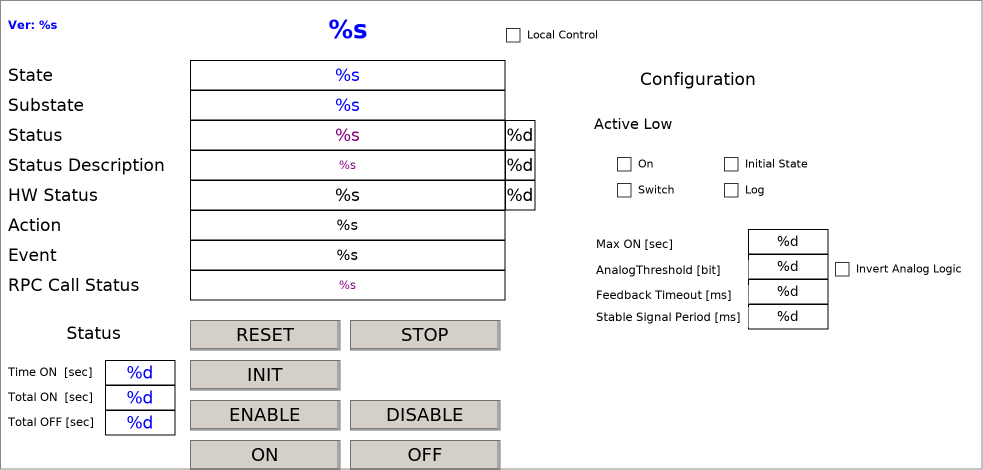
VISUALIZATION GUI_TEMPLATE_ACTUATOR  // 983x470
VAR_IN_OUT
	m_Instance:	FB_ACTUATOR;
END_VAR
    Rectangle (190,60 315x30), "%s", text variable: m_Instance.stat.sState
    Rectangle (190,90 315x30), "%s", text variable: m_Instance.stat.sSubstate
    Button (190,320 150x30), "RESET", input disabled if: (m_Instance.stat.bLocal = FALSE) <> 0
        OnMouseDown: execute { m_Instance.ctrl.nCommand := E_ACTUATOR_COMMAND.RESET; m_Instance.ctrl.bExecute := TRUE; }
    Button (190,360 150x30), "INIT", input disabled if: (m_Instance.stat.bLocal = FALSE) <> 0
        OnMouseDown: execute { m_Instance.ctrl.nCommand := E_ACTUATOR_COMMAND.INIT; m_Instance.ctrl.bExecute := TRUE; }
    Button (350,320 150x30), "STOP", input disabled if: (m_Instance.stat.bLocal = FALSE) <> 0
        OnMouseDown: execute { m_Instance.ctrl.nCommand := E_ACTUATOR_COMMAND.STOP; m_Instance.ctrl.bExecute := TRUE; }
    Button (190,400 150x30), "ENABLE", input disabled if: (m_Instance.stat.bLocal = FALSE) <> 0
        OnMouseDown: execute { m_Instance.ctrl.nCommand := E_ACTUATOR_COMMAND.ENABLE; m_Instance.ctrl.bExecute := TRUE; }
    Button (350,400 150x30), "DISABLE", input disabled if: (m_Instance.stat.bLocal = FALSE) <> 0
        OnMouseDown: execute { m_Instance.ctrl.nCommand := E_ACTUATOR_COMMAND.DISABLE; m_Instance.ctrl.bExecute := TRUE; }
    Button (190,440 150x30), "ON", input disabled if: (m_Instance.stat.bLocal = FALSE) <> 0
        OnMouseDown: execute { m_Instance.ctrl.nCommand := E_ACTUATOR_COMMAND.ON; m_Instance.ctrl.bExecute := TRUE; }
    Button (350,440 150x30), "OFF", input disabled if: (m_Instance.stat.bLocal = FALSE) <> 0
        OnMouseDown: execute { m_Instance.ctrl.nCommand := E_ACTUATOR_COMMAND.OFF; m_Instance.ctrl.bExecute := TRUE; }
    Rectangle (5,60 180x30), "State"
    Rectangle (5,90 180x30), "Substate"
    Rectangle (190,120 315x30), "%s", text variable: m_Instance.stat.sStatus
    Rectangle (190,150 315x30), "%s", text variable: m_Instance.stat.sErrorText
    Rectangle (5,120 180x30), "Status"
    Rectangle (5,150 180x30), "Status Description"
    Rectangle (190,210 315x30), "%s", text variable: m_Instance.stat.sActionDesc
    Rectangle (190,240 315x30), "%s", text variable: m_Instance.stat.sEventDesc
    Rectangle (190,180 315x30), "%s", text variable: m_Instance.stat.sHwStatus
    Rectangle (5,180 180x30), "HW Status"
    Rectangle (505,180 30x30), "%d", text variable: m_Instance.stat.nHwStatus
    Rectangle (5,210 180x30), "Action"
    Rectangle (5,240 180x30), "Event"
    Rectangle (232,12 232x35), "%s", text variable: m_Instance.cfg.sName
    Rectangle (637,64 180x30), "Configuration"
    Rectangle (591,109 126x30), "Active Low"
    Checkbox (615,149 72x30), "On", variable: m_Instance.cfg.bActiveLowOn, input disabled if: (m_Instance.stat.bLocal = FALSE) <> 0
    Checkbox (615,175 72x30), "Switch", variable: m_Instance.cfg.bActiveLowSwitch, input disabled if: (m_Instance.stat.bLocal = FALSE) <> 0
    Checkbox (833,254 150x30), "Invert Analog Logic", tooltip "If the logic is inverted, the actuator is considered to be ON, if the reading is below the threshold.", variable: m_Instance.cfg.bInvertAnalog, input disabled if: (m_Instance.stat.bLocal = FALSE) <> 0
    Rectangle (593,234 155x20), "Max ON [sec]"
    Rectangle (748,229 80x25), "%d", tooltip "Maximum allowed time for actuator to be ON [sec] (>=0). Zero means no limit.", text variable: m_Instance.cfg.nMaxOn, input disabled if: (m_Instance.stat.bLocal = FALSE) <> 0
        OnMouseDown: write the text variable via Default, min 0
    Rectangle (748,254 80x25), "%d", tooltip "Analog feedback signal threshold [bit]. If used, the threshold should be > 0.", text variable: m_Instance.cfg.nAnalogThreshold, input disabled if: (m_Instance.stat.bLocal = FALSE) <> 0
        OnMouseDown: write the text variable via Default, min 0
    Rectangle (593,260 155x20), "AnalogThreshold [bit]"
    Rectangle (748,279 80x25), "%d", tooltip "When switching actuator ON, feedback signal should become active within this period.", text variable: m_Instance.cfg.nTimeout, input disabled if: (m_Instance.stat.bLocal = FALSE) <> 0
        OnMouseDown: write the text variable via Default, min 0
    Rectangle (593,285 155x20), "Feedback Timeout [ms]"
    Checkbox (504,20 116x30), "Local Control", variable: m_Instance.stat.bLocal
    Rectangle (748,304 80x25), "%d", tooltip "A period of time [ms] that the feedback signal has to have constant value before taking its status. Minimum 10 ms.", text variable: m_Instance.cfg.nSigStablePeriod, input disabled if: (m_Instance.stat.bLocal = FALSE) <> 0
        OnMouseDown: write the text variable via Default, min 10
    Rectangle (593,307 155x20), "Stable Signal Period [ms]"
    Rectangle (48,318 92x30), "Status"
    Rectangle (105,360 70x25), "%d", tooltip "Time since last ON command [sec].", text variable: m_Instance.stat.nTimeOn
    Rectangle (105,385 70x25), "%d", tooltip "Total continuous time that actuator has been ON [sec].", text variable: m_Instance.stat.nTimeOnTotal
    Rectangle (105,410 70x25), "%d", tooltip "Time since actuator was switched OFF [sec].", text variable: m_Instance.stat.nTimeOff
    Rectangle (5,357 95x30), "Time ON [sec]"
    Rectangle (5,382 95x30), "Total ON [sec]"
    Rectangle (5,407 95x30), "Total OFF [sec]"
    Rectangle (505,120 30x30), "%d", text variable: m_Instance.stat.nStatus
    Rectangle (190,270 315x30), "%s", text variable: m_Instance.stat.sRPCErrorText
    Rectangle (5,270 180x30), "RPC Call Status"
    Rectangle (5,10 99x30), "Ver: %s", tooltip "'Actuator.library version'", text variable: stLibVersion_ESO_LDC_Actuator_Library.sVersion, input disabled if: true
    Checkbox (722,175 72x30), "Log", tooltip "If checked, logging is active.", variable: m_Instance.cfg.bLog, input disabled if: (m_Instance.stat.bLocal = FALSE) <> 0
    Checkbox (722,149 107x30), "Initial State", tooltip "If checked, switch is automatically turned ON on PLC reboot or after RESET.", variable: m_Instance.cfg.bInitialState, input disabled if: (m_Instance.stat.bLocal = FALSE) <> 0
    Rectangle (505,150 30x30), "%d", tooltip "Error code. Zero means no error.", text variable: m_Instance.stat.nErrorCode
END_VISUALIZATION

(* stored: Version 1.1.0.1, ProductVersion 3.1.4024.3
   Visu GUI_TEMPLATE_ACTUATOR: Id {208abcb1-f1a3-4a00-92a5-f362cd7556ac} *)
